INTERFACE I_Motor

PROPERTY bAuto : BOOL
GET
END_GET
SET
END_SET
END_PROPERTY

PROPERTY bEnable : BOOL
GET
END_GET
SET
END_SET
END_PROPERTY

PROPERTY bRunning : BOOL
GET
END_GET
END_PROPERTY

PROPERTY nSpeed : INT
GET
END_GET
SET
END_SET
END_PROPERTY

END_INTERFACE

(* stored: Version 1.1.0.1
   Itf I_Motor: Id {4d969e27-ae96-48de-93d6-06a00a18b9d7}
   Property bAuto: Id {ae5c7314-fccf-4c52-9f44-fe72b00a6070}
   Get Get: Id {c3806af1-7510-49dd-9ee2-568278bf5d68}
   Set Set: Id {27360742-a540-4e99-b72c-7181fa019906}
   Property bEnable: Id {fdd803ef-7c3a-4993-b978-eb4399925c4e}
   Get Get: Id {d14bd4f5-10b2-4a18-a17a-0d8aeb80e795}
   Set Set: Id {25671867-117e-4e39-bef0-2138bb2f5346}
   Property bRunning: Id {36f8461c-674f-4e9c-94b1-b2799b049781}
   Get Get: Id {7e6b71aa-efc0-4c14-bae6-639eddbf76a0}
   Property nSpeed: Id {1b9f1cc0-8438-4c22-a52c-75b0388d68fd}
   Get Get: Id {f55835ad-359a-463a-9c3e-bba3564f1341}
   Set Set: Id {ce1ea666-8437-4c96-9cdd-0a9d4e9e7081} *)
